PROGRAM MAIN
VAR
	Initialize	:	BOOL := TRUE;
	
	AttemptReset : TON := (PT:=T#500ms);
    
    DisplayStats : FB_CXSetTextDisplayUSB := (nPort:=28928);
    fbFormat   : FB_FormatString;
    bError     : BOOL;
    nErrID     : UDINT;
    sOut       : T_MaxString;   
    
	fbLogHandler : FB_LogHandler;
	fbEcatDiag : FB_EcatDiagWrapper;

	{attribute 'pytmc' := '
		pv: Arbiter:Link:HGVPU
		link: USEG:UNDH:
	'}
	fbHgvpu : FB_Hgvpu;
	
	{attribute 'pytmc' := '
		pv: Arbiter:Link:SXU
		link: USEG:UNDS:
	'}
	fbSxu : FB_SXU;
	
END_VAR

//Arbiter PLC

IF Initialize THEN
	Initialize := FALSE;
END_IF

MachineSimulation();
		
PMPS_Arbiter();

AttemptReset(IN:=GVL.g_FastFaultOutput1.xOK, Q=>GVL.g_FastFaultOutput1.i_xReset);

(*
DisplayStats.bExecute S= NOT DisplayStats.bBusy AND NOT DisplayStats.bError;
DisplayStats.bExecute R= DisplayStats.bBusy OR DisplayStats.bError;

DisplayStats.sLine1 := 'PMPS-ARBITER-K';
fbFormat(sFormat := 'Fast Faults: %d', arg1:=F_ULINT(PMPS_GVL.AccumulatedFF), sOut=>DisplayStats.sLine2, bError => bError, nErrID => nErrID ); 

DisplayStats(eMode:=E_CX2100_DisplayModesWr.eCX2100_WriteLines);
*)

fbEcatDiag();
fbLogHandler();

ACTION Initialize:

END_ACTION

END_PROGRAM

(* stored: Version 1.1.0.1, ProductVersion 3.1.4022.18
   POU MAIN: Id {8a7bcfd2-1a2b-4363-aa47-c19391bf1f9c}, SpecialFunc None
   Action Initialize: Id {b0ee480a-3d4b-001d-04c4-43cdc47895c8} *)
